FUNCTION_BLOCK FB_DigitalSensNC
VAR_INPUT
	_input	: BOOL;
END_VAR

VAR_OUTPUT
	_output : BOOL;
END_VAR

_output := NOT _input;

PROPERTY IsActive : BOOL
GET
IsActive:= _output;
END_GET
END_PROPERTY

END_FUNCTION_BLOCK

(* stored: Version 1.1.0.1, ProductVersion 3.1.4024.16
   POU FB_DigitalSensNC: Id {bc8c9ce5-05eb-43da-a6ef-61809be1250e}, SpecialFunc None
   Property IsActive: Id {8a6a15d5-0eeb-4501-90c4-2aa077e15e25}
   Get Get: Id {b609fe4a-581c-4e60-bed0-a275fdba00d6} *)
